INTERFACE ITF_Object

PROPERTY Index : int
GET
END_GET
SET
END_SET
END_PROPERTY

END_INTERFACE

(* stored: Version 1.1.0.1, ProductVersion 3.1.4024.11
   Itf ITF_Object: Id {2b0b3e0f-86b8-4a58-808e-487231f944d3}
   Property Index: Id {304f8c06-1551-4318-8628-aa3a5da2f156}
   Get Get: Id {6a0576db-67fc-4ffa-9d3b-538d89a4a887}
   Set Set: Id {8cd099b0-beb2-440a-8836-3a651c2f23f6} *)
